{attribute 'qualified_only'}
{attribute 'strict'}
TYPE ERetargetType :
(
	not_retargeted := 0,
	primitive_target := 1,
	sequence_target := 2
);
END_TYPE

(* stored: Version 1.1.0.1
   DUT ERetargetType: Id {d67be642-fb09-4163-8835-ef0fed7a4c5c} *)
